(* IEC 61131-3 sources: ArfBotOS/Codesys-4/ArfBotOS.fbsdev/Application.iecapp^/FUN/template/FB_PackML.fb.st^, 3 files *)

(* ---- M_Execute.meth.st ---- *)
METHOD PROTECTED M_Execute : BOOL
VAR_INPUT
END_VAR
END_METHOD

(* ---- M_SetPackML.meth.st ---- *)
METHOD PROTECTED M_SetPackML : BOOL
VAR_INPUT
END_VAR

_UnitMode(sName := 'Normal Operation',
			dwSupportedStates := PACK_ML.State.All,
			dwAllowsLeavingFromStates := PACK_ML.State.Stopped
											OR PACK_ML.State.Aborted
											OR PACK_ML.State.Idle,
			dwAllowsEnteringIntoStates := PACK_ML.State.Stopped
											OR PACK_ML.State.Aborted
											OR PACK_ML.State.Idle,
			eInitialState := PACK_ML.State.Idle,
			xActive := TRUE);
END_METHOD

(* ---- M_StateComplete.meth.st ---- *)
METHOD PROTECTED M_StateComplete : BOOL
VAR_INPUT
END_VAR

_UnitMode.ActingStateCompleted();
END_METHOD
